// TIA Portal V17 export
// export: Created 2024-08-07T21:43:55.3634139Z, ExportSetting WithDefaults, DisplayName Totally Integrated Automation Portal, DisplayVersion V17 Update 7, DisplayName TIA Portal Openness, DisplayVersion V17 Update 7, DisplayName TIA Portal Version Control Interface, DisplayVersion V17, DisplayName SINAMICS Startdrive Advanced, DisplayVersion V17 SP2, DisplayName SINAMICS Startdrive G110M, G120, G120C, G120D, G120P, G115D, DisplayVersion V17 SP2, DisplayName SINAMICS Startdrive G130, G150, S120, S150, SINAMICS MV, S210, DisplayVersion V17 SP2, DisplayName STEP 7 Professional, DisplayVersion V17 Update 7, DisplayName STEP 7 Safety, DisplayVersion V17 Update 6, DisplayName WinCC Advanced / Unified PC, DisplayVersion V17 Update 7
DATA_BLOCK "FittingHistoryLeftCupforming_DB"   // DB35
VERSION : 0.1
// stored: AutoNumber true, DBAccessibleFromOPCUA true, DBAccessibleFromWebserver true, InstanceOfName FittingHistory, InstanceOfType FB
"FittingHistory"
   // VAR_INPUT
   //    iNewCycle : Bool;
   //    iData : "UDT_Results_Cupforming";
   // END_VAR
   // VAR RETAIN
   //    history : Array[0..99] of "UDT_Results_Cupforming";
   // END_VAR
   // VAR
   //    pageData { S7_SetPoint := 'True'} : Array[0..9] of "UDT_Results_Cupforming";
   // END_VAR
   // VAR RETAIN
   //    pageNumber { S7_SetPoint := 'True'} : USInt := 0;
   // END_VAR
   // VAR
   //    resetHistory : Bool;
   //    R_TRIG_Instance { S7_SetPoint := 'True'} : R_TRIG;
   // END_VAR
BEGIN
   history[0].MaxForce := -7.98946;
   history[1].MaxForce := -7.998657;
   history[2].MaxForce := -7.98946;
   history[3..4].MaxForce := -7.984862;
   history[5].MaxForce := -8.007853;
   history[6].MaxForce := -7.994059;
   history[7].MaxForce := -7.980264;
   history[8].MaxForce := 32.33566;
   history[9].MaxForce := 30.64817;
   history[10].MaxForce := 27.33296;
   history[11..99].MaxForce := 0.0;
   history[0].MinimalWay := 9.841429;
   history[1].MinimalWay := 9.875875;
   history[2].MinimalWay := 9.837013;
   history[3].MinimalWay := 9.846728;
   history[4].MinimalWay := 9.887358;
   history[5].MinimalWay := 9.779602;
   history[6].MinimalWay := 9.831714;
   history[7].MinimalWay := 9.859094;
   history[8].MinimalWay := 8.49007;
   history[9].MinimalWay := 8.491837;
   history[10].MinimalWay := 8.488304;
   history[11..99].MinimalWay := 0.0;
   history[0].MaxZposition := 55.44488;
   history[1].MaxZposition := 55.55556;
   history[2].MaxZposition := 55.54471;
   history[3].MaxZposition := 55.3928;
   history[4].MaxZposition := 55.42969;
   history[5].MaxZposition := 55.67492;
   history[6].MaxZposition := 55.59462;
   history[7].MaxZposition := 55.36676;
   history[8].MaxZposition := 59.20356;
   history[9].MaxZposition := 59.29688;
   history[10].MaxZposition := 59.16667;
   history[11..99].MaxZposition := 0.0;
   history[0..10].OK := TRUE;
   history[11..99].OK := FALSE;
   history[0..99].NOK := FALSE;
   history[0..10].parameters.DigiforceProgram := 1;
   history[11..99].parameters.DigiforceProgram := 0;
   history[0..10].parameters.FinalSpeed := 20.0;
   history[11..99].parameters.FinalSpeed := 0.0;
   history[0..10].parameters.ApproachSpeed := 100.0;
   history[11..99].parameters.ApproachSpeed := 0.0;
   history[0..7].parameters.FinalForce := 80.0;
   history[8..10].parameters.FinalForce := 90.0;
   history[11..99].parameters.FinalForce := 0.0;
   history[0..10].parameters.ApproachForce := 20.0;
   history[11..99].parameters.ApproachForce := 0.0;
   history[0..7].parameters.EndWayImmediate := 9.9;
   history[8..10].parameters.EndWayImmediate := 8.5;
   history[11..99].parameters.EndWayImmediate := 0.0;
   history[0..7].parameters.EndWayWithTimeout := 9.9;
   history[8..9].parameters.EndWayWithTimeout := 8.6;
   history[10].parameters.EndWayWithTimeout := 8.5;
   history[11..99].parameters.EndWayWithTimeout := 0.0;
   history[0..7].parameters.SwitchingWay := 50.0;
   history[8..10].parameters.SwitchingWay := 53.0;
   history[11..99].parameters.SwitchingWay := 0.0;
   history[0..10].parameters.EndWayTimeout := T#300MS;
   history[11..99].parameters.EndWayTimeout := T#0MS;
END_DATA_BLOCK
